% RSLogix 500 project I2P JOB 12 - FORWARD-REVERSE USING SS OF 1P MOTOR_BAK010.RSS, saved by version 10.00.00.00 %
PROJECT "ML6A"    % processor: Bul.1763 MicroLogix 1100 Series B %

PROGRAM FILES
  LAD 2   5 rungs

DATA FILES
  O0 OUTPUT  4 elements
  I1 INPUT  6 elements
  S2 STATUS  66 elements
  B3 BINARY  1 elements
  T4 TIMER  1 elements
  C5 COUNTER  1 elements
  R6 CONTROL  1 elements
  N7 INTEGER  1 elements
  F8 FLOAT  1 elements

LADDER 2
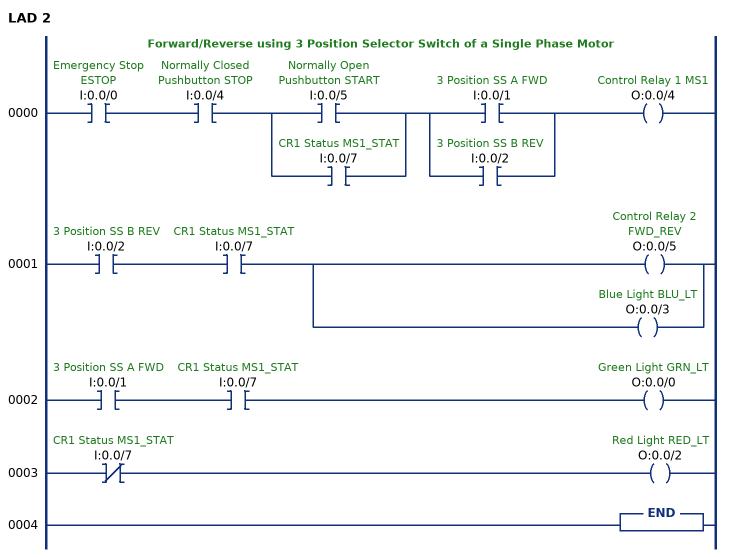
% Rung: 0 %
% TITLE: Forward/Reverse using 3 Position Selector Switch of a Single Phase Motor %
SOR XIC I:0.0/0 XIC I:0.0/4 BST XIC I:0.0/5 NXB XIC I:0.0/7 BND BST XIC I:0.0/1 NXB XIC I:0.0/2 BND OTE O:0.0/4 EOR
%   I:0.0/0  ESTOP  "Emergency Stop" %
%   I:0.0/4  STOP  "Normally Closed Pushbutton" %
%   I:0.0/5  START  "Normally Open Pushbutton" %
%   I:0.0/7  MS1_STAT  "CR1 Status" %
%   I:0.0/1  FWD  "3 Position SS A" %
%   I:0.0/2  REV  "3 Position SS B" %
%   O:0.0/4  MS1  "Control Relay 1" %
% Rung: 1 %
SOR XIC I:0.0/2 XIC I:0.0/7 BST OTE O:0.0/5 NXB OTE O:0.0/3 BND EOR
%   I:0.0/2  REV  "3 Position SS B" %
%   I:0.0/7  MS1_STAT  "CR1 Status" %
%   O:0.0/5  FWD_REV  "Control Relay 2" %
%   O:0.0/3  BLU_LT  "Blue Light" %
% Rung: 2 %
SOR XIC I:0.0/1 XIC I:0.0/7 OTE O:0.0/0 EOR
%   I:0.0/1  FWD  "3 Position SS A" %
%   I:0.0/7  MS1_STAT  "CR1 Status" %
%   O:0.0/0  GRN_LT  "Green Light" %
% Rung: 3 %
SOR XIO I:0.0/7 OTE O:0.0/2 EOR
%   I:0.0/7  MS1_STAT  "CR1 Status" %
%   O:0.0/2  RED_LT  "Red Light" %
% Rung: 4 %
SOR END EOR

OTHER DOCUMENTED ADDRESSES
  I:0.0/3  2PSS  "2 Position SS"
  I:0.0/6  PB3  "Normally Open Pushbutton"
  I:0.0/8  CR2_STAT  "CR2 Status"
  O:0.0/1  YLW_LT  "Yellow Light"
